// TIA Portal project "Pick and Place V2" (V17)

(* hardware
DEVICE "S7-300/ET200M station_1"  S7-300 station
   slot 0: "Rail_0"  Rail  6ES7 390-1***0-0AA0
   slot 1: "PS 307 5A_1"  PS 307 5A  6ES7 307-1EA00-0AA0
   slot 2: "PLC_1"  CPU 315F-2 PN/DP  6ES7 315-2FH13-0AB0  V2.6
      slot 1: "MPI/DP interface_1"  X1
      slot 2: "PROFINET interface_1"  PN-IO
         slot 1: "Port_1"  Port
   slot 4: "DI 16/DO 16x24VDC/0.5A_1"  DI16/DO16 x 24V / 0.5A  6ES7 323-1BL00-0AA0
   slot 5: "AI 4/AO 2x8BIT_1"  AI4/AO2 x 8 bits  6ES7 334-0CE01-0AA0
   slot 6: "DI 8/DO 8x24VDC/0.5A_1"  DI8/DO8 x 24VDC / 0.5A  6ES7 323-1BH01-0AA0
*)

// ===== PLC "PLC_1"  CPU 315F-2 PN/DP =====

VAR_GLOBAL   // PLC tag table "Default tag table"
   "RB_Aan" AT %Q0.0 : Bool;   // Rolband aan of uit mono
   "ZN_N_Binnen" AT %Q0.1 : Bool;   // Zuignap beweegst naar binnen
   "ZN_N_Buiten" AT %Q0.2 : Bool;   // Zuignap beweegst naar Buiten
   "ZN_N_Beneden" AT %Q0.3 : Bool;   // Zuignap beweegst omlaag (Mono
   "ZN_T_Vacuum" AT %Q0.4 : Bool;   // Zuignap trekt Vacuum
   "CP_S_RB" AT %Q0.5 : Bool;   // Inverse mono halverwege checkpoint
   "S_Lading" AT %Q0.7 : Bool;   // Signaal naar vorig station
   "D_Lading_Voor" AT %I0.0 : Bool;   // Detectie lading vooraan
   "D_Lading_CP" AT %I0.4 : Bool;   // Detectie lading halverwege
   "D_ZN_Vacuum" AT %I0.3 : Bool;   // Detectie Vacuum getrokken
   "D_ZN_Hoog" AT %I0.5 : Bool;   // Detectie Zuignap boven
   "D_ZN_Buiten" AT %I0.2 : Bool;   // Detectie Zuignap Buiten
   "D_ZN_Binnen" AT %I0.1 : Bool;   // Detectie Zuignap Binnen
   "Timer_Lossen" AT %T0 : Timer;   // Timer 2 sec lossen lading
   "D_M_Lading" AT %M0.0 : Bool;
END_VAR

DATA_BLOCK "Main_Safety_RTG1_DB"   // DB1, F_DB
{ S7_Optimized_Access := 'FALSE' }
VERSION : 0.1
// stored: InstanceOfName Main_Safety_RTG1
"Main_Safety_RTG1"
BEGIN
END_DATA_BLOCK

DATA_BLOCK "Block_2_DB"   // DB2
{ S7_Optimized_Access := 'FALSE' }
VERSION : 0.1
// stored: InstanceOfName Block_2
"Block_2"
BEGIN
END_DATA_BLOCK

FUNCTION_BLOCK "Main_Safety_RTG1"   // FB1, F_LAD
{ S7_Optimized_Access := 'FALSE' }
BEGIN
END_FUNCTION_BLOCK

FUNCTION_BLOCK "Block_2"   // FB2, GRAPH
{ S7_Optimized_Access := 'FALSE' }
VERSION : 0.1
   VAR_INPUT
      OFF_SQ : Bool := false;   // Turn sequence off
      INIT_SQ : Bool := false;   // Set sequence to initial state
      ACK_EF : Bool := false;   // Acknowledge all errors and faults
      S_PREV : Bool := false;   // Output previous step in parameter S_NO
      S_NEXT : Bool := false;   // Indicate next step in parameter S_NO
      SW_AUTO : Bool := false;   // Automatic mode
      SW_TAP : Bool := false;   // Semiautomatic/switch with transition
      SW_TOP : Bool := false;   // Semiautomatic/ignore transition
      SW_MAN : Bool := false;   // Manual mode
      S_SEL : Int := 0;   // Select step to be output to S_NO
      S_ON : Bool := false;   // Activate step indicated in S_NO
      S_OFF : Bool := false;   // Deactivate step indicated S_NO
      T_PUSH : Bool := false;   // Enable transition to switch in semi automatic mode
   END_VAR
   VAR_OUTPUT
      S_NO : Int := 0;   // Step number
      S_MORE : Bool := false;   // More steps are available and can be shown in S_NO
      S_ACTIVE : Bool := false;   // Step indicated in S_NO is active
      ERR_FLT : Bool := false;   // Interlock or supervision group error
      AUTO_ON : Bool := false;   // Automatic mode is active
      TAP_ON : Bool := false;   // Semiautomatic mode/step with transition enabled
      TOP_ON : Bool := false;   // Semiautomatic mode/ignore transition enabled
      MAN_ON : Bool := false;   // Manual mode is active
   END_VAR
   VAR
      SWITCH : Array[0..0] of DWord;
      SW_SQTS : Array[0..10] of Byte;
      SW_ADDR : Word := 16#A;
      G7T_0 : GraphTransition;
      G7S_0 : GraphStep;
      PRE_CRIT : Array[0..0] of DWord;
      POST_CRIT : Array[0..0] of DWord;
      TVX : Array[0..2] of Byte;
      TTX : Array[0..2] of Byte;
      TSX : Array[0..2] of Byte;
      S00X : Array[0..2] of Byte;
      SOFFX : Array[0..2] of Byte;
      SONX : Array[0..2] of Byte;
      SAX : Array[0..2] of Byte;
      SERRX : Array[0..11] of Byte;
      SMX : Array[0..11] of Byte;
      S0X : Array[0..11] of Byte;
      S1X : Array[0..11] of Byte;
      S_DISPLAY : Int;   // Internal display of output parameter S_NO
      S_SEL_OLD : Int;   // Previous value in S_SEL
      S_DISPIDX : Byte;   // Index of the step in S_NO
      T_DISPIDX : Byte;   // Index of the transition displayed in T_NO
      MOPEDGE : Struct
         AUTO : Bool := false;
         MAN : Bool := false;
         TAP : Bool := false;
         TOP : Bool := false;
         ACK_S : Bool := false;
         REG_S : Bool := false;
         T_PREV : Bool := false;
         T_NEXT : Bool := false;
         LOCK : Bool := false;
         SUP : Bool := false;
         ACKREQ : Bool := false;
         SSKIP : Bool := false;
         OFF : Bool := false;
         INIT : Bool := false;
         HALT : Bool := false;
         TMS_HALT : Bool := false;
         OPS_ZERO : Bool := false;
         SACT_DISP : Bool := false;
         SEF_DISP : Bool := false;
         SALL_DISP : Bool := false;
         S_PREV : Bool := false;
         S_NEXT : Bool := false;
         S_SELOK : Bool := false;
         S_ON : Bool := false;
         S_OFF : Bool := false;
         T_PUSH : Bool := false;
         REG : Bool := false;
         ACK : Bool := false;
         IL_PERM : Bool := false;
         T_PERM : Bool := false;
         ILP_MAN : Bool := false;
      END_STRUCT;
      MOP : Struct   // Mode
         AUTO : Bool := true;   // Status: automatic mode
         MAN : Bool := false;   // Status: manual mode
         TAP : Bool := false;   // Status: semi automatic/switch with transition
         TOP : Bool := false;   // Status: semi automatic/ignore transition
         ACK_S : Bool := false;   // Request: acknowledge step at parameter S_NO
         REG_S : Bool := false;   // Request: register step indicated in S_NO
         T_PREV : Bool := false;   // Request: output previous valid transition in T_NO
         T_NEXT : Bool := false;   // Request: output next valid transition in T_NO
         LOCK : Bool := true;   // Status: interlocks activated
         SUP : Bool := true;   // Status: supervisions activated
         ACKREQ : Bool := true;   // Status: acknowledgment required
         SSKIP : Bool := false;   // Status: "Skip steps" enabled
         OFF : Bool := false;   // Request: deactivate all steps
         INIT : Bool := true;   // Request: set sequence to initial state
         HALT : Bool := false;   // Status: sequence halted
         TMS_HALT : Bool := false;   // Status: all internal timers held
         OPS_ZERO : Bool := false;   // Status: set all operands processed with N, L, D instructions to 0
         SACT_DISP : Bool := true;   // Status: display active steps only
         SEF_DISP : Bool := false;   // Status: display only steps with errors and disrupted steps
         SALL_DISP : Bool := false;   // Status: display all steps
         S_PREV : Bool := false;   // Request: output previous step to S_NO
         S_NEXT : Bool := false;   // Request: Output next step at S_NO parameter
         S_SELOK : Bool := false;   // Request: output step number from S_SEL to S_NO
         S_ON : Bool := false;   // Request: activate step indicated in S_NO
         S_OFF : Bool := false;   // Request: deactivate step at parameter S_NO
         T_PUSH : Bool := false;   // Request: transition switching enabled
         REG : Bool := false;   // Request: register all interlock and supervision errors
         ACK : Bool := false;   // Request: acknowledge all interlock and supervision errors
         IL_PERM : Bool := false;   // Status: permanent processing of all interlocks
         T_PERM : Bool := false;   // Status: permanent processing of all transitions
         ILP_MAN : Bool := false;   // Status: permanent processing of all interlocks in manual mode
      END_STRUCT;
      TICKS : Struct   // Clock speeds
         DELTA : Time := T#0ms;   // Time difference between cycles
         OLD : Time := T#0ms;   // 10 ms clock counter value in last cycle
         NEW : Time := T#0ms;   // 10 ms clock counter value in this cycle
      END_STRUCT;
      SQ_FLAGS : Struct   // Sequence bit memory
         ERR_FLT : Bool := false;   // Interlock and supervision group error
         ERROR : Bool := false;   // Interlock group error
         FAULT : Bool := false;   // Supervision group error
         RT_FAIL : Bool := false;   // Runtime error
         NO_SNO : Bool := false;   // Requested step number not found
         NF_OFL : Bool := false;   // Overflow: too many ON or OFF requests
         SA_OFL : Bool := false;   // Overflow: too many steps active
         TV_OFL : Bool := false;   // Overflow: too many valid transitions
         MSG_OFL : Bool := false;   // Overflow: not enough system resources for ALARM_S
         NO_SWI : Bool := false;   // Do not switch in this cycle
         CYC_OP : Bool := false;   // Cyclic execution of the sequence after initialization
         AS_MSG : Bool := true;   // Alarms during runtime enabled or disabled by instruction
         AS_SEND : Bool := false;   // Send alarms from WR_USMSG or only enter in diagnostics buffer
         SQ_BUSY : Bool := false;   // Internal edge bit memory for sequence processing
         SA_BUSY : Bool := false;   // Internal edge bit memory for sequence processing
         AS_SIG : Bool := false;   // Edge bit memory for alarms from Alarm_S and Alarm_SQ
      END_STRUCT;
      S_PTR : DWord := 16#660;
      S_PTR2 : DWord := 16#0;
      S_PTR3 : DWord := 16#13A0;
      S_PTR4 : DWord := 16#1340;
      T_PTR : DWord := 16#12E0;
      C_AR2 : DWord := 16#0;
      M_FBDB : DWord := 16#20000;
      M_SNO : Word := 16#0;
      M_EVID : Word := 16#0;
      M_EVIL : C_Alarm_s;
      M_EVSV : C_Alarm_s;
      M_EV : DWord := 16#1220;
      CRIT : Array[0..31] of Bool;
      S_START : Byte := 16#0;
      S_IDX : Byte := 16#0;
      S_INT : Int := 72;
      S_TMP : Byte := 16#0;
      T_START : Byte := 16#0;
      T_IDX : Byte := 16#0;
      T_TMP : Byte := 16#0;
      T_TMP2 : Byte := 16#00;
      TV_POT : Byte := 16#06;
      RETURN1 : Byte := 16#0;
      RETURN2 : Byte := 16#0;
      SINI : Array[0..2] of Byte;
      LSTT : Array[0..10] of Byte;
      ATAJ : Array[0..10] of Byte;
      ATAB : Array[0..10] of Byte;
      PSTT : Array[0..10] of Byte;
      NSTT : Array[0..10] of Byte;
      ASSJ : Array[0..10] of Byte;
      ASSB : Array[0..10] of Byte;
      PTTS : Array[0..10] of Byte;
      NTTS : Array[0..10] of Byte;
      PRE_CNT : Word := 16#1;
      POST_CNT : Word := 16#1;
      ADR_COND : Word := 16#0;
      MAX_TVAL : Byte := 16#1;
      MAX_SACT : Byte := 16#1;
      MAX_CRIT : Byte := 16#4;
      T_CNT : Byte := 16#A;
      SUP_CNT : Byte := 16#0;
      LOCK_CNT : Byte := 16#0;
      S_CNT : Byte := 16#A;
      SQ_CNT : Byte := 16#1;
      PRS_INPAR : DWord := 16#E000FEC8;
      PRS_OUTPAR : DWord := 16#E000800F;
      GC_FLAGS : Struct
         T_MACH : Byte := 16#EB;
         COND_ED : Byte := 16#E3;
         W_LEVEL : Byte := 16#D5;
         FB_IF : Byte := 16#FA;
         AS_MSG : Word := 16#404;
         SSB : Word := 16#108;
         DILG : Word := 16#370;
         ADDR_T0 : Word := 16#1C;
         CRIT_AVAIL : Bool := false;
         SSKIP_AVAIL : Bool := true;
         SSKIP_ON : Bool := false;
         ACK_REQ : Bool := true;
         SYNC_AVAIL : Bool := true;
         ILP_MAN : Bool := false;
         SWM_LOCKED : Bool := false;
         SAVE_SW : Bool := true;
      END_STRUCT;
      G7_FBMARK : Byte := 16#3C;
      G7_RELEASE : Byte := 16#3C;
      G7_ID2 : Byte := 16#37;
      G7_ID1 : Byte := 16#47;
   END_VAR
   // SW_SQTS[0] := 16#1;
   // TVX[0] := 16#1;
   // TTX[0] := 16#1;
   // TSX[0] := 16#1;
   // S00X[0] := 16#1;
   // SOFFX[0] := 16#1;
   // SONX[0] := 16#1;
   // SAX[0] := 16#1;
   // SERRX[0] := 16#1;
   // SMX[0] := 16#1;
   // S0X[0] := 16#1;
   // S1X[0] := 16#1;
   // SINI[0] := 16#2;
   // SINI[1] := 16#1;
   // SINI[2] := 0;
   // LSTT[0] := 0;
   // LSTT[1] := 0;
   // LSTT[2] := 0;
   // LSTT[3] := 0;
   // LSTT[4] := 0;
   // LSTT[5] := 0;
   // LSTT[6] := 0;
   // LSTT[7] := 0;
   // ATAJ[0] := 0;
   // ATAJ[1] := 16#1;
   // ATAJ[2] := 16#2;
   // ATAJ[3] := 16#3;
   // ATAJ[4] := 16#4;
   // ATAJ[5] := 16#5;
   // ATAJ[6] := 16#6;
   // ATAJ[7] := 16#7;
   // ATAB[0] := 0;
   // ATAB[1] := 16#1;
   // ATAB[2] := 16#2;
   // ATAB[3] := 16#3;
   // ATAB[4] := 16#4;
   // ATAB[5] := 16#5;
   // ATAB[6] := 16#6;
   // ATAB[7] := 16#7;
   // PSTT[0] := 0;
   // PSTT[1] := 16#1;
   // PSTT[2] := 16#2;
   // PSTT[3] := 16#3;
   // PSTT[4] := 16#4;
   // PSTT[5] := 16#5;
   // PSTT[6] := 16#6;
   // PSTT[7] := 16#7;
   // NSTT[0] := 16#1;
   // NSTT[1] := 16#2;
   // NSTT[2] := 16#3;
   // NSTT[3] := 16#4;
   // NSTT[4] := 16#5;
   // NSTT[5] := 16#6;
   // NSTT[6] := 16#7;
   // NSTT[7] := 16#8;
   // ASSJ[0] := 0;
   // ASSJ[1] := 16#1;
   // ASSJ[2] := 16#2;
   // ASSJ[3] := 16#3;
   // ASSJ[4] := 16#4;
   // ASSJ[5] := 16#5;
   // ASSJ[6] := 16#6;
   // ASSJ[7] := 16#7;
   // ASSB[0] := 0;
   // ASSB[1] := 16#1;
   // ASSB[2] := 16#2;
   // ASSB[3] := 16#3;
   // ASSB[4] := 16#4;
   // ASSB[5] := 16#5;
   // ASSB[6] := 16#6;
   // ASSB[7] := 16#7;
   // PTTS[0] := 0;
   // PTTS[2] := 16#1;
   // PTTS[3] := 16#2;
   // PTTS[4] := 16#3;
   // PTTS[5] := 16#4;
   // PTTS[6] := 16#5;
   // PTTS[7] := 16#6;
   // NTTS[0] := 0;
   // NTTS[1] := 16#1;
   // NTTS[2] := 16#2;
   // NTTS[3] := 16#3;
   // NTTS[4] := 16#4;
   // NTTS[5] := 16#5;
   // NTTS[6] := 16#6;
   // NTTS[7] := 16#7;
   // LSTT[8] := 0;
   // LSTT[9] := 0;
   // LSTT[10] := 16#1;
   // ATAJ[8] := 16#8;
   // ATAJ[9] := 16#9;
   // ATAJ[10] := 16#A;
   // ATAB[8] := 16#8;
   // ATAB[9] := 16#9;
   // ATAB[10] := 16#A;
   // PSTT[8] := 16#8;
   // PSTT[9] := 16#9;
   // PSTT[10] := 16#A;
   // NSTT[8] := 16#9;
   // NSTT[9] := 16#A;
   // NSTT[10] := 16#1;
   // ASSJ[8] := 16#8;
   // ASSJ[9] := 16#9;
   // ASSJ[10] := 16#A;
   // ASSB[8] := 16#8;
   // ASSB[9] := 16#9;
   // ASSB[10] := 16#A;
   // PTTS[8] := 16#7;
   // PTTS[9] := 16#8;
   // PTTS[10] := 16#9;
   // NTTS[8] := 16#8;
   // NTTS[9] := 16#9;
   // NTTS[10] := 16#A;
BEGIN
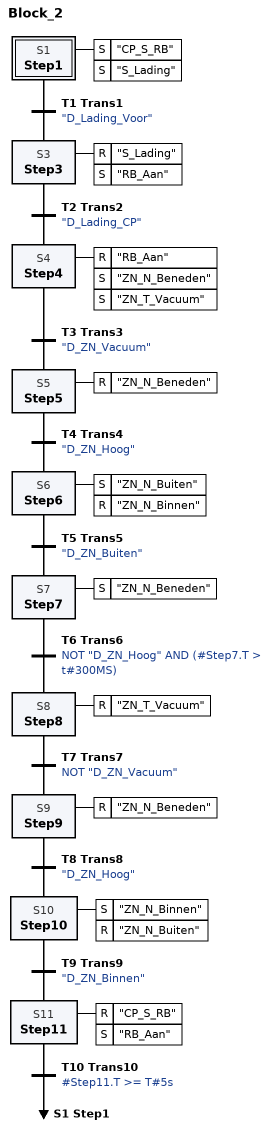
   // sequencer 1
   INITIAL_STEP Step1:   // S1
              S    "CP_S_RB"
              S    "S_Lading"
   END_STEP
   TRANSITION Trans1 FROM Step1 TO Step3   // T1
      := "D_Lading_Voor";
   END_TRANSITION
   STEP Step3:   // S3
              R    "S_Lading"
              S    "RB_Aan"
   END_STEP
   TRANSITION Trans2 FROM Step3 TO Step4   // T2
      := "D_Lading_CP";
   END_TRANSITION
   STEP Step4:   // S4
              R    "RB_Aan"
              S    "ZN_N_Beneden"
              S    "ZN_T_Vacuum"
   END_STEP
   TRANSITION Trans3 FROM Step4 TO Step5   // T3
      := "D_ZN_Vacuum";
   END_TRANSITION
   STEP Step5:   // S5
              R    "ZN_N_Beneden"
   END_STEP
   TRANSITION Trans4 FROM Step5 TO Step6   // T4
      := "D_ZN_Hoog";
   END_TRANSITION
   STEP Step6:   // S6
              S    "ZN_N_Buiten"
              R    "ZN_N_Binnen"
   END_STEP
   TRANSITION Trans5 FROM Step6 TO Step7   // T5
      := "D_ZN_Buiten";
   END_TRANSITION
   STEP Step7:   // S7
              S    "ZN_N_Beneden"
   END_STEP
   TRANSITION Trans6 FROM Step7 TO Step8   // T6
      := NOT "D_ZN_Hoog" AND (#Step7.T > t#300MS);
   END_TRANSITION
   STEP Step8:   // S8
              R    "ZN_T_Vacuum"
   END_STEP
   TRANSITION Trans7 FROM Step8 TO Step9   // T7
      := NOT "D_ZN_Vacuum";
   END_TRANSITION
   STEP Step9:   // S9
              R    "ZN_N_Beneden"
   END_STEP
   TRANSITION Trans8 FROM Step9 TO Step10   // T8
      := "D_ZN_Hoog";
   END_TRANSITION
   STEP Step10:   // S10
              S    "ZN_N_Binnen"
              R    "ZN_N_Buiten"
   END_STEP
   TRANSITION Trans9 FROM Step10 TO Step11   // T9
      := "D_ZN_Binnen";
   END_TRANSITION
   STEP Step11:   // S11
              R    "CP_S_RB"
              S    "RB_Aan"
   END_STEP
   TRANSITION Trans10 FROM Step11 TO Step1   // T10, jump
      := #Step11.T >= T#5s;
   END_TRANSITION
END_FUNCTION_BLOCK

ORGANIZATION_BLOCK "Main"   // OB1, LAD
TITLE = "Main Program Sweep (Cycle)"
{ S7_Optimized_Access := 'FALSE' }
VERSION : 0.1
   VAR_TEMP
      OB1_EV_CLASS : Byte;   // Bits 0-3 = 1 (Coming event), Bits 4-7 = 1 (Event class 1)
      OB1_SCAN_1 : Byte;   // 1 (Cold restart scan 1 of OB 1), 3 (Scan 2-n of OB 1)
      OB1_PRIORITY : Byte;   // Priority of OB Execution
      OB1_OB_NUMBR : Byte;   // 1 (Organization block 1, OB1)
      OB1_RESERVED_1 : Byte;   // Reserved for system
      OB1_RESERVED_2 : Byte;   // Reserved for system
      OB1_PREV_CYCLE : Int;   // Cycle time of previous OB1 scan (milliseconds)
      OB1_MIN_CYCLE : Int;   // Minimum cycle time of OB1 (milliseconds)
      OB1_MAX_CYCLE : Int;   // Maximum cycle time of OB1 (milliseconds)
      OB1_DATE_TIME : Date_And_Time;   // Date and time OB1 started
   END_VAR
BEGIN

REGION Network 1
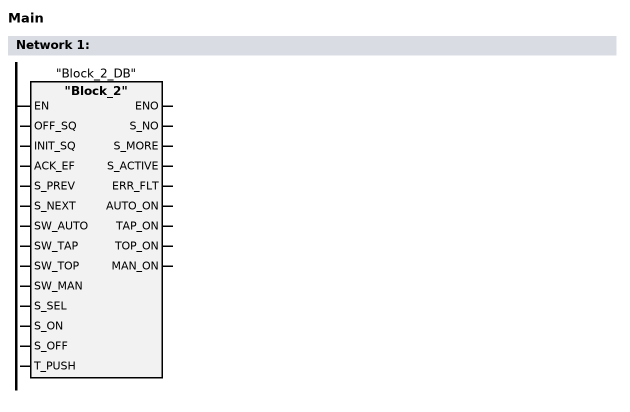
   RUNG wire#powerrail
      "Block_2_DB"(OFF_SQ :=, INIT_SQ :=, ACK_EF :=, S_PREV :=, S_NEXT :=, SW_AUTO :=, SW_TAP :=, SW_TOP :=, SW_MAN :=, S_SEL :=, S_ON :=, S_OFF :=, T_PUSH :=, S_NO =>, S_MORE =>, S_ACTIVE =>, ERR_FLT =>, AUTO_ON =>, TAP_ON =>, TOP_ON =>, MAN_ON =>)
   END_RUNG
   // the same network as SCL:
   "Block_2_DB"();   // "Block_2"
END_REGION
END_ORGANIZATION_BLOCK

ORGANIZATION_BLOCK "CYC_INT5_RTG1"   // OB35, LAD
TITLE = "Cyclic Interrupt"
{ S7_Optimized_Access := 'FALSE' }
VERSION : 0.1
   VAR_TEMP
      OB35_EV_CLASS : Byte;   // Bits 0-3 = 1 (Coming event), Bits 4-7 = 1 (Event class 1)
      OB35_STRT_INF : Byte;   // 16#36 (OB 35 has started)
      OB35_PRIORITY : Byte;   // Priority of OB Execution
      OB35_OB_NUMBR : Byte;   // 35 (Organization block 35, OB35)
      OB35_RESERVED_1 : Byte;   // Reserved for system
      OB35_RESERVED_2 : Byte;   // Reserved for system
      OB35_PHASE_OFFSET : Word;   // Phase offset (msec)
      OB35_RESERVED_3 : Int;   // Reserved for system
      OB35_EXC_FREQ : Int;   // Frequency of execution (msec)
      OB35_DATE_TIME : Date_And_Time;   // Date and time OB35 started
   END_VAR
BEGIN

REGION Network 1
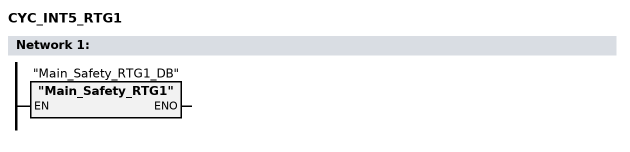
   RUNG wire#powerrail
      "Main_Safety_RTG1_DB"()
   END_RUNG
   // the same network as SCL:
   "Main_Safety_RTG1_DB"();   // "Main_Safety_RTG1"
END_REGION
END_ORGANIZATION_BLOCK